// TIA Portal V20 export
TYPE "typeGaugeRnRHmiInterface"
// stored: Access Published, Namespace Unit1.Em8
   STRUCT
      currentCount : Int;
      processCount : Int := 50;
   END_STRUCT;
END_TYPE
